FUNCTION_BLOCK fb_motor
VAR_INPUT
	bStart, bStop : BOOL;
	
END_VAR
VAR_OUTPUT
	bStatus : BOOL;
END_VAR
VAR
END_VAR

END_FUNCTION_BLOCK

(* stored: Version 1.1.0.1, ProductVersion 3.1.4024.11
   POU fb_motor: Id {0ebc1963-e29c-4f87-83f3-c3853d7fd186}, SpecialFunc None *)
